TYPE (* ISOBUS UT position-marker object pool properties (Change Child Position child/parent + travel bounds + center offset) *)
  (* Standard: 61499-2; Description: Copyright (c) 2026 Meisterschulen am Ostbahnhof This program and the accompanying materials are made available under the terms of the Eclipse Public License 2.0 which is available at https://www.eclipse.org/legal/epl-2.0/ SPDX-License-Identifier: EPL-2.0 *)
  (* Version 1.0, 2026-09-05, Franz Höpfinger, Meisterschulen am Ostbahnhof, initial API and implementation and/or initial documentation *)
  PACKAGE isobus::utils::childposition;
  IMPORT isobus::UT::Q::const::IDs;
  PositionMarker_S : STRUCT
    u16ChildId : UINT := IDs::ID_NULL; (* Object ID of the moved VT object (Change Child Position child, e.g. a CPolygon) *)
    u16ParentId : UINT := IDs::ID_NULL; (* Object ID of the parent VT container the child moves within (Change Child Position parent) *)
    r32MinPos : REAL := 0.0; (* Lower bound of the child's valid X-travel inside the parent, in raw pixels (normally 0.0) *)
    r32MaxPos : REAL := 0.0; (* Upper bound of the child's valid X-travel inside the parent, in raw pixels = ContainerWidth - ChildBoundingBoxWidth *)
    r32Center : REAL := 0.0; (* Offset added to the incoming value before clamping - the raw pixel X position that corresponds to value = 0.0 *)
    s16YPosition : INT := 0; (* Fixed Y position passed straight through to Q_ChildPosition.s16Yposition (this FB drives only the X axis) *)
  END_STRUCT;
END_TYPE
